// TIA Portal V21 export
DATA_BLOCK "__PI_CREATEDB_NAME__"   // DB__PI_CREATEDB_NUMBER__
{ S7_Optimized_Access := 'TRUE' }
// Minimal disposable global DB template imported by TiaLocalBridge.
// stored: MemoryReserve 100
BEGIN
END_DATA_BLOCK
